// Mitsubishi GX Works2 project: Time Control   PLC: Q03UDV

PROGRAM MAIN
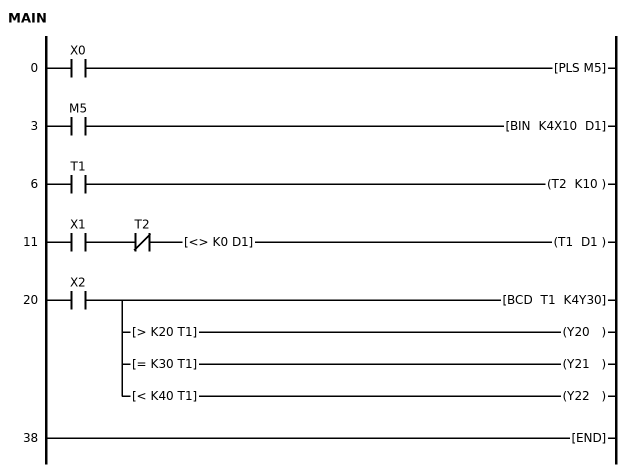
0     LD      X0
      PLS     M5
3     LD      M5
      BIN     K4X10 D1
6     LD      T1
      OUT     T2 K10
11    LD      X1
      ANI     T2
      AND<>   K0 D1
      OUT     T1 D1
20    LD      X2
      BCD     T1 K4Y30
      MPS
      AND>    K20 T1
      OUT     Y20
      MRD
      AND=    K30 T1
      OUT     Y21
      MPP
      AND<    K40 T1
      OUT     Y22
38    END
END_PROGRAM
